Yaskawa INFORM job: SKRZYNIA_4040_180_STOPNI_10B_OLD.JBI

/JOB
//NAME SKRZYNIA_4040_180_STOPNI_10B_OLD
///FOLDERNAME 02-SKRZYNIE_JOBS
//POS
///NPOS 593,593,0,24,0,0
///TOOL 0
///POSTYPE PULSE
///PULSE
C00000=-21231,-51303,42314,2367,6591,-1439
C00001=-12854,-61498,-6635,149088,-29435,16513
C00002=84284,-61498,-6635,149088,14842,16513
C00003=84426,-61498,-62039,149088,14842,16513
C00004=84426,-61498,-83719,149088,14842,16513
C00005=40079,-25830,-61904,72398,37828,17494
C00006=40079,-25830,-61904,72398,37828,17494
C00007=38824,-23395,-60038,72349,38727,17731
C00008=41545,-22667,-59464,70826,37145,18191
C00009=40079,-25830,-61904,72398,37828,17494
C00010=40079,-23879,-31232,97616,36989,2612
C00011=40241,-22903,-30855,97033,36795,2952
C00012=39596,-21803,-29985,96678,37187,3182
C00013=41542,-21522,-29763,96797,35874,3054
C00014=40241,-22903,-30855,97033,36795,2952
C00015=32191,-51498,-15746,88434,42441,22641
C00016=44500,-22967,-34027,49689,40772,15208
C00017=44759,-21950,-33222,49364,40770,15399
C00018=43898,-20603,-32137,49608,41392,15289
C00019=45676,-20288,-31878,48567,40497,15854
C00020=44759,-21950,-33222,49364,40770,15399
C00021=50639,-31838,-53853,40430,42590,20636
C00022=47737,-42531,-47731,84740,46626,-3202
C00023=73324,-51450,-15857,136644,48513,-27329
C00024=28578,-31257,-33285,101874,54895,-3139
C00025=29101,-23166,-41439,93785,52323,3372
C00026=30342,-16402,-40775,90158,51109,6027
C00027=29555,-14242,-38855,90054,51607,6222
C00028=31304,-14182,-38798,89754,50458,6198
C00029=30342,-16402,-40775,90158,51109,6027
C00030=37840,-26567,-47806,97824,39338,5403
C00031=38314,-22656,-45541,96192,38787,6352
C00032=38740,-21749,-44817,95954,38481,6451
C00033=38106,-20505,-43805,95701,38856,6673
C00034=39920,-20274,-43616,95549,37666,6573
C00035=38740,-21749,-44817,95954,38481,6451
C00036=35154,-23288,-28184,89821,43405,2441
C00037=35403,-21021,-26397,89340,43215,2751
C00038=34678,-19569,-25213,89063,43699,2948
C00039=36545,-19419,-25091,89018,42427,2940
C00040=35403,-21021,-26397,89340,43215,2751
C00041=46673,-28267,-59493,36306,49500,22578
C00042=47298,-25083,-54483,36432,48421,22382
C00043=46134,-23276,-53085,36983,49197,22170
C00044=48093,-22778,-52692,35651,48513,22818
C00045=47298,-25083,-54483,36432,48421,22382
C00046=43000,-32780,-49011,53703,41088,15214
C00047=66148,-65994,-55487,105361,28212,-7739
C00048=66148,-65994,-55487,105361,28212,-7739
C00049=59848,-54778,-49507,133915,29212,-10807
C00050=45497,-38347,-41839,114412,32622,-465
C00051=46376,-32635,-46933,102993,29107,5780
C00052=46303,-28031,-46898,97061,28371,8976
C00053=45038,-26161,-45521,96183,29128,9541
C00054=46946,-25787,-45238,96120,27855,9431
C00055=46303,-28031,-46898,97061,28371,8976
C00056=45864,-17128,1685,129467,40696,-9274
C00057=46023,-15894,1830,128891,40053,-8896
C00058=45181,-14790,2774,128176,40341,-8535
C00059=46921,-14545,2986,129317,39465,-9073
C00060=45402,-17127,796,128656,40504,-8810
C00061=42828,-21985,-11573,106778,34538,-1929
C00062=43349,-21404,-11124,106831,34165,-1930
C00063=42250,-19876,-9917,105946,34757,-1485
C00064=44494,-19460,-9583,106781,33302,-1837
C00065=42797,-21858,-11474,106726,34550,-1903
C00066=72417,-67880,-88171,46465,42262,31903
C00067=72417,-67880,-88171,46465,42262,31903
C00068=81480,-74508,-67932,111005,17511,3722
C00069=42492,-36415,-29790,92406,42740,11684
C00070=29699,-14901,-14062,86637,51249,15251
C00071=28921,-12904,-12269,86425,51786,15406
C00072=30978,-12767,-12144,86426,50380,15429
C00073=29506,-17416,-16239,86937,51377,15018
C00074=88410,-69609,-60867,139529,19008,-8209
C00075=62412,-62489,-12046,-12266,17816,34850
C00076=0,-52280,40443,0,6876,0
C00077=-681,-52632,38645,-5695,5489,-631
C00078=-17840,-61498,-6635,-149088,-29435,-16513
C00079=-84284,-61498,-6635,-149088,14842,-16513
C00080=-84426,-61498,-62039,-149088,14842,-16513
C00081=-84426,-61498,-83719,-149088,14842,-16513
C00082=-83351,-27062,-60322,-167360,37385,6517
C00083=-83351,-27062,-60322,-167360,37385,23281
C00084=-45097,-23850,-79932,-76262,26943,-22849
C00085=-48253,-15729,-73342,-71138,25693,-24842
C00086=-50302,-13076,-73239,-65836,25323,-27140
C00087=-49401,-11675,-71961,-66260,25816,-27133
C00088=-50608,-11574,-71867,-65226,25249,-27391
C00089=-49660,-13361,-73494,-66442,25615,-26975
C00090=-48242,-21102,-77802,-73044,25430,-23851
C00091=-42432,-29691,-46140,-101591,34194,-3953
C00092=-40467,-32259,-45349,-89481,35752,-6083
C00093=-35590,-22323,-38089,-87474,43148,-7978
C00094=-34853,-20780,-36847,-87247,43643,-8181
C00095=-37029,-20471,-36594,-86926,42180,-8224
C00096=-35503,-23333,-38886,-87700,43207,-7835
C00097=-41659,-25848,-37197,-61468,39541,-12344
C00098=-42019,-23363,-32043,-63110,38591,-11327
C00099=-41283,-22167,-31102,-63128,39154,-11341
C00100=-43189,-21868,-30866,-62281,38009,-11788
C00101=-40846,-25460,-35158,-62968,39555,-11455
C00102=-39561,-32409,-42051,-71473,38885,-9254
C00103=-88477,-67032,-53890,-125185,13082,17955
C00104=-90715,-66667,-50935,-152816,24533,28486
C00105=-30735,-26920,-32844,-95116,50209,-1071
C00106=-37180,-24683,-31930,-114741,47007,2943
C00107=-36407,-19634,-34656,-109847,45004,-453
C00108=-38352,-16604,-33863,-108521,43129,-1176
C00109=-37479,-14809,-32279,-108169,43576,-1482
C00110=-39395,-14487,-31992,-108361,42368,-1194
C00111=-37253,-18321,-35339,-108644,43916,-1187
C00112=-30948,-19486,-27368,-89515,49970,-2899
C00113=-32453,-17458,-25663,-89179,48933,-3088
C00114=-31896,-16151,-24534,-89028,49305,-3221
C00115=-33527,-16125,-24510,-88960,48196,-3202
C00116=-31291,-18911,-26892,-89421,49733,-2955
C00117=-32789,-14788,-10714,-75998,48642,-1904
C00118=-33953,-13481,-9550,-75758,47902,-2112
C00119=-33380,-12226,-8408,-75670,48319,-2157
C00120=-35020,-12164,-8351,-75529,47228,-2306
C00121=-33300,-14767,-10697,-75957,48300,-1949
C00122=-33300,-14767,-10697,-75957,48300,-1949
C00123=-33901,-13199,-7224,-76945,47663,-1266
C00124=-33178,-11617,-5779,-76815,48184,-1329
C00125=-35129,-11426,-5603,-76688,46886,-1497
C00126=-32900,-14718,-9841,-76444,48459,-1584
C00127=-46324,-38325,-53351,-48650,39022,-16558
C00128=-84678,-53272,-42524,-56273,5220,-14251
C00129=-79949,-57830,-54545,-43165,18800,-25262
C00130=-85199,-63426,-59279,-35356,8253,-25340
C00131=-43240,-40066,-69296,-76804,34492,-13950
C00132=-32352,-24302,-62495,-76398,48702,-17646
C00133=-33867,-19497,-59989,-74208,48202,-18898
C00134=-33043,-17469,-58279,-74274,48770,-19034
C00135=-35172,-17180,-58031,-73305,47532,-19251
C00136=-33150,-20833,-61090,-74721,48572,-18687
C00137=-32525,-19963,-22291,-97454,48417,-2656
C00138=-34479,-17146,-19937,-97221,47013,-2812
C00139=-33716,-15515,-18525,-96928,47480,-3025
C00140=-35357,-15455,-18472,-97073,46375,-2908
C00141=-33341,-18474,-21063,-97306,47817,-2759
C00142=-32838,-10388,7981,-94473,48357,2926
C00143=-33747,-9461,8037,-94117,47673,2571
C00144=-33094,-8062,9377,-93861,48090,2458
C00145=-34952,-7927,9507,-94260,46861,2543
C00146=-33010,-10379,7174,-94037,48174,2591
C00147=-74406,-60637,-53290,-78600,32734,-4861
C00148=-74406,-60637,-53290,-78600,32734,-4861
C00149=-66351,-49775,-22313,-121187,42752,19491
C00150=-38126,-18978,-6321,-103556,42156,4232
C00151=-39485,-17529,-8330,-90200,39091,223
C00152=-38315,-15563,-6658,-89669,39866,-39
C00153=-40130,-15376,-6497,-89855,38637,-21
C00154=-40610,-23081,-12745,-91737,38407,1092
C00155=-82794,-45547,-18103,-153793,26453,27163
///LIMIT ON
C00156=-46099,-67236,-11725,-98004,28606,19827
C00157=275,-40498,62911,330,272,-175
///LIMIT OFF
C00158=-21231,-51303,42314,2367,6591,-1439
C00159=-12854,-61498,-6635,149088,-29435,16513
C00160=84284,-61498,-6635,149088,14842,16513
C00161=84426,-61498,-62039,149088,14842,16513
C00162=84426,-61498,-83719,149088,14842,16513
C00163=40079,-25830,-61904,72398,37828,17494
C00164=43542,-21744,-53414,85694,32141,12908
C00165=43538,-20959,-59091,78847,32551,16732
C00166=40079,-23879,-31232,97616,36989,2612
C00167=41069,-22296,-36683,87871,35939,7163
C00168=41069,-20857,-27994,94343,36275,3375
C00169=40241,-22903,-30855,97033,36795,2952
C00170=44500,-22967,-34027,49689,40772,15208
C00171=37674,-14410,-29425,54908,51799,12689
C00172=37617,-13106,-20810,58248,49229,10178
C00173=44759,-21950,-33222,49364,40770,15399
C00174=50639,-31838,-53853,40430,42590,20636
C00175=47737,-42531,-47731,84740,46626,-3202
C00176=78714,-49092,-28755,133609,38199,-24420
C00177=28578,-31257,-33285,101874,54895,-3139
C00178=29101,-23166,-41439,93785,52323,3372
C00179=31163,-13872,-34138,92103,50752,4440
C00180=31163,-14064,-41434,88282,50498,7326
C00181=30342,-16402,-40775,90158,51109,6027
C00182=37840,-26567,-47806,97824,39338,5403
C00183=38314,-22656,-45541,96192,38787,6352
C00184=39658,-19881,-39017,99036,38353,4498
C00185=39658,-20227,-46296,93241,37598,7980
C00186=38740,-21749,-44817,95954,38481,6451
C00187=35154,-23288,-28184,89821,43405,2441
C00188=36302,-20456,-32356,81251,42995,6506
C00189=36302,-19046,-24537,85721,42698,3608
C00190=35403,-21021,-26397,89340,43215,2751
C00191=46673,-28267,-59493,36306,49500,22578
C00192=35383,-14910,-45807,52457,59655,19882
C00193=35383,-15025,-38926,54776,56903,17744
C00194=47298,-25083,-54483,36432,48421,22382
C00195=43000,-32780,-49011,53703,41088,15214
C00196=90538,-65158,-52413,145953,6697,-22013
C00197=90538,-65158,-52413,145953,6697,-22013
C00198=59848,-54778,-49507,133915,29212,-10807
C00199=45497,-38347,-41839,114412,32622,-465
C00200=46376,-32635,-46933,102993,29107,5780
C00201=38443,-20223,-37840,96971,39567,10287
C00202=38443,-20698,-44956,91660,38993,13539
C00203=46303,-28031,-46898,97061,28371,8976
C00204=45864,-17128,1685,129467,40696,-9274
C00205=38069,-7942,12691,120284,49952,-5070
C00206=38069,-11604,1369,116685,47266,-2469
C00207=45402,-17127,796,128656,40504,-8810
C00208=42828,-21985,-11573,106778,34538,-1929
C00209=33281,-15275,-13406,92642,47209,4970
C00210=33281,-12456,-2996,97026,47894,1870
C00211=42797,-21858,-11474,106726,34550,-1903
C00212=72417,-64226,-72669,53660,37323,27470
C00213=81480,-74508,-67932,111005,17511,3722
C00214=31559,-23192,-27729,97069,50041,14774
C00215=34278,-17590,-29530,108925,47275,14558
C00216=34921,-13948,-26935,108215,46513,15013
C00217=34921,-14719,-34056,104413,45059,17611
C00218=33936,-16225,-25259,110400,48238,13526
C00219=30729,-14807,-22031,91030,50318,16982
C00220=30729,-13019,-13516,94566,50766,14318
C00221=88410,-69609,-60867,139529,19008,-8209
C00222=62412,-62489,-12046,-12266,17816,34850
C00223=0,-52280,40443,0,6876,0
C00224=-681,-52632,38645,-5695,5489,-631
C00225=-17840,-61498,-6635,-149088,-29435,-16513
C00226=-84284,-61498,-6635,-149088,14842,-16513
C00227=-84426,-61498,-62039,-149088,14842,-16513
C00228=-84426,-61498,-83719,-149088,14842,-16513
C00229=-83351,-27062,-60322,-167360,37385,6517
C00230=-83351,-27062,-60322,-167360,37385,23281
C00231=-45097,-23850,-79932,-76262,26943,-22849
C00232=-48253,-15729,-73342,-71138,25693,-24842
C00233=-42869,-6204,-67496,-75794,33821,-25861
C00234=-42869,-3205,-70686,-69723,34977,-29338
C00235=-49660,-13361,-73494,-66442,25615,-26975
C00236=-48242,-21102,-77802,-73044,25430,-23851
C00237=-42432,-29691,-46140,-101591,34194,-3953
C00238=-40467,-32259,-45349,-89481,35752,-6083
C00239=-32032,-15700,-34761,-86363,49905,-9645
C00240=-32032,-14866,-27372,-89947,49973,-6979
C00241=-35503,-23333,-38886,-87700,43207,-7835
C00242=-41659,-25848,-37197,-61468,39541,-12344
C00243=-32550,-13183,-23016,-68651,53358,-8526
C00244=-34023,-12481,-22084,-63241,53452,-9524
C00245=-40846,-25460,-35158,-62968,39555,-11455
C00246=-39561,-32409,-42051,-71473,38885,-9254
C00247=-88477,-67032,-53890,-125185,13082,17955
C00248=-90715,-66667,-50935,-152816,24533,28486
C00249=-30735,-26920,-32844,-95116,50209,-1071
C00250=-37180,-24683,-31930,-114741,47007,2943
C00251=-36407,-19634,-34656,-109847,45004,-453
C00252=-39264,-14095,-28560,-110319,43249,69
C00253=-39254,-14742,-35710,-105973,41627,-2729
C00254=-37253,-18321,-35339,-108644,43916,-1187
C00255=-30948,-19486,-27368,-89515,49970,-2899
C00256=-33188,-17217,-33290,-80523,49125,-7157
C00257=-33231,-16133,-25752,-84153,48705,-4513
C00258=-31291,-18911,-26892,-89421,49733,-2955
C00259=-32789,-14788,-10714,-75998,48642,-1904
C00260=-32456,-10000,-8763,-74569,51725,-2878
C00261=-32456,-7502,814,-78111,50801,-165
C00262=-33300,-14767,-10697,-75957,48300,-1949
C00263=-33300,-14767,-10697,-75957,48300,-1949
C00264=-31039,-7597,-4415,-75714,54029,-1891
C00265=-31745,-5891,1281,-74609,53027,-1007
C00266=-32900,-14718,-9841,-76444,48459,-1584
C00267=-46324,-38325,-53351,-48650,39022,-16558
C00268=-84678,-53272,-42524,-56273,5220,-14251
C00269=-79949,-57830,-54545,-43165,18800,-25262
C00270=-85199,-63426,-59279,-35356,8253,-25340
C00271=-43240,-40066,-69296,-76804,34492,-13950
C00272=-32352,-24302,-62495,-76398,48702,-17646
C00273=-34311,-15084,-43386,-89458,46770,-12174
C00274=-34303,-14562,-49859,-85086,46777,-15220
C00275=-33150,-20833,-61090,-74721,48572,-18687
C00276=-32525,-19963,-22291,-97454,48417,-2656
C00277=-35706,-13608,-12356,-102024,46946,-662
C00278=-35706,-15621,-21438,-97808,45877,-3577
C00279=-33341,-18474,-21063,-97306,47817,-2759
C00280=-32838,-10388,7981,-94473,48357,2926
C00281=-33093,-7396,5806,-90907,49596,566
C00282=-33114,-3922,16616,-94789,50065,3444
C00283=-33010,-10379,7174,-94037,48174,2591
C00284=-73757,-59015,-49060,-81128,30370,-3444
C00285=-66351,-49775,-22313,-115582,40632,19491
C00286=-39230,-13378,9505,-118180,46878,7841
C00287=-45382,-7236,12023,-133378,48537,9962
C00288=-45404,-10871,608,-130166,44845,7725
C00289=-39289,-13633,5656,-114159,44810,6160
C00290=-38323,-13232,3563,-106275,42852,3854
C00291=-39624,-12309,2722,-105485,41613,3229
C00292=-39624,-8328,14658,-110578,43519,6514
C00293=-36264,-16485,7382,-110054,45980,6615
C00294=-44249,-32643,-4456,-118298,43922,12613
C00295=-31781,-48654,10305,-108801,40875,18482
///LIMIT ON
C00296=275,-40498,62911,330,272,-175
///LIMIT OFF
C00297=-21231,-51303,42314,2367,6591,-1439
C00298=-12854,-61498,-6635,149088,-29435,16513
C00299=32880,-72586,-50560,79734,53940,25582
C00300=76664,-93599,-96338,114349,24908,7990
C00301=72545,-76403,-90681,98079,12187,16258
C00302=68435,-42241,-79282,43384,21203,43145
C00303=65057,-16377,-54230,51764,24572,24912
C00304=65057,-16377,-54230,51764,24572,24912
C00305=63338,-14509,-52578,53100,25585,24479
C00306=65493,-13068,-51269,50530,24633,25485
C00307=65057,-16377,-54230,51764,24572,24912
C00308=65057,-15356,-24189,99795,20011,765
C00309=64877,-14372,-23690,98704,20045,1316
C00310=64002,-13489,-22890,98156,20604,1621
C00311=65592,-12702,-22173,98357,19527,1466
C00312=64877,-14372,-23690,98704,20045,1316
C00313=68341,-13254,-25781,29903,31229,25524
C00314=68283,-12212,-24821,29865,31356,25548
C00315=67188,-11145,-23825,30867,31841,25051
C00316=68624,-10377,-23095,29361,31405,25809
C00317=68283,-12212,-24821,29865,31356,25548
C00318=67373,-28813,-51747,26561,36937,27500
C00319=65665,-56911,-59086,75825,31170,1181
C00320=86238,-56758,-47218,93606,16664,-7096
C00321=86238,-56758,-47218,93606,16664,-7096
C00322=58162,-25487,-29222,106212,35121,-6052
C00323=54729,-17550,-36821,90686,35172,3055
C00324=53879,-10723,-35593,84994,35691,6442
C00325=52628,-8898,-33837,85063,36512,6546
C00326=54193,-8333,-33282,84633,35489,6620
C00327=53879,-10723,-35593,84994,35691,6442
C00328=63265,-18185,-41125,95483,22448,4389
C00329=62561,-14368,-38517,92984,22773,5727
C00330=62689,-13396,-37636,92694,22678,5861
C00331=61812,-12400,-36718,92465,23238,6064
C00332=63331,-11679,-36046,92201,22238,6052
C00333=62689,-13396,-37636,92694,22678,5861
C00334=60836,-16142,-22303,87853,25853,3109
C00335=60346,-13901,-20318,87240,26185,3441
C00336=59279,-12702,-19226,86999,26911,3593
C00337=60868,-12050,-18626,86765,25831,3679
C00338=60346,-13901,-20318,87240,26185,3441
C00339=71174,-16943,-50501,16787,44328,31924
C00340=70846,-13961,-45205,17496,43056,31510
C00341=69412,-12602,-43961,18675,43507,30969
C00342=70949,-11616,-43043,17320,43301,31610
C00343=70846,-13961,-45205,17496,43056,31510
C00344=66765,-25643,-43957,33958,30926,25005
C00345=89904,-51519,-74342,14421,36812,44678
C00346=59533,-60921,-66479,83565,41795,11392
C00347=74572,-27669,-34920,136415,14797,-11887
C00348=72479,-21736,-38943,108586,11547,1590
C00349=70901,-17325,-38411,94105,11830,8638
C00350=69318,-15905,-37172,92885,12849,9347
C00351=70820,-15051,-36412,92531,11846,9399
C00352=70901,-17325,-38411,94105,11830,8638
C00353=70927,-7523,10343,151197,29871,-19432
C00354=70517,-6236,10737,150221,29352,-18933
C00355=69462,-5331,11645,148944,29606,-18324
C00356=70849,-4645,12343,150548,29173,-19084
C00357=70402,-7634,9356,150158,29478,-18907
C00358=68660,-13051,-4106,122816,18275,-8999
C00359=68895,-12351,-3471,122899,18094,-9031
C00360=67458,-11121,-2337,120787,18802,-8043
C00361=69212,-10147,-1425,122703,17774,-8922
C00362=68590,-12934,-4000,122687,18305,-8939
C00363=75423,-38775,-29488,68062,11357,11878
C00364=75423,-38775,-29488,68062,11357,11878
C00365=83800,-53438,-37305,103753,25026,-1265
C00366=73693,-43023,-29306,101200,31062,8332
C00367=57182,-8361,13896,122065,42938,1264
C00368=54175,-4244,10116,111777,38351,4895
C00369=53015,-2664,11762,111180,39035,5172
C00370=54334,-2350,12093,111780,38228,4906
C00371=54175,-4244,10116,111777,38351,4895
C00372=89016,-59505,-36896,143842,20811,-11822
C00373=0,-52280,40443,0,6876,0
C00374=-681,-52632,38645,-5695,5489,-631
C00375=-17840,-61498,-6635,-149088,-29435,-16513
C00376=-84284,-61498,-6635,-149088,14842,-16513
C00377=-57949,-92832,-68327,-119114,39180,-13331
C00378=-51160,-78996,-68705,-103851,38676,-21739
C00379=-70129,-12201,-70194,-45988,15849,-32683
C00380=-70861,-4247,-62448,-43170,16032,-33903
C00381=-72229,-1292,-61598,-37253,16795,-36501
C00382=-71164,-286,-60510,-39045,17142,-35862
C00383=-72168,114,-60071,-37345,16819,-36474
C00384=-71747,-1710,-62044,-38091,16943,-36199
C00385=-72086,-8949,-67137,-41785,15362,-34318
C00386=-68226,-19972,-38714,-103620,16923,-1218
C00387=-67549,-22986,-38612,-80975,17520,-9124
C00388=-60286,-14955,-31870,-81576,26630,-9634
C00389=-59206,-13694,-30736,-81541,27366,-9725
C00390=-61026,-12796,-29913,-80837,26167,-9971
C00391=-60502,-15936,-32740,-81790,26471,-9505
C00392=-66711,-16726,-29834,-42060,26790,-21996
C00393=-66477,-14329,-24475,-44917,25565,-20507
C00394=-65503,-13376,-23611,-45716,26132,-20127
C00395=-67048,-12587,-22889,-44009,25442,-20959
C00396=-66009,-16611,-27996,-44380,26285,-20808
C00397=-67084,-23473,-35621,-52822,22843,-18344
C00398=-54372,-63877,-56403,-90862,27079,1323
C00399=-55608,-75012,-34654,-126966,55573,20814
C00400=-55608,-75012,-34654,-126966,55573,20814
C00401=-58069,-20780,-28125,-95622,31565,-134
C00402=-62818,-16895,-25617,-123146,31403,8811
C00403=-60301,-12189,-28106,-114654,29999,4030
C00404=-61167,-8731,-26593,-112607,28768,2985
C00405=-59960,-7252,-25135,-111997,29446,2563
C00406=-61574,-6413,-24296,-112502,28453,2957
C00407=-60636,-10677,-28466,-112685,29164,2987
C00408=-55814,-13636,-22293,-87541,33030,-3263
C00409=-56566,-11270,-20110,-87077,32519,-3496
C00410=-55709,-10167,-19066,-86969,33101,-3589
C00411=-57154,-9687,-18605,-86794,32120,-3632
C00412=-55949,-12989,-21706,-87412,32939,-3330
C00413=-57109,-8613,-4995,-71756,32687,-5152
C00414=-57764,-7017,-3429,-71410,32292,-5358
C00415=-56909,-5946,-2356,-71529,32873,-5273
C00416=-58347,-5433,-1836,-71115,31941,-5534
C00417=-57555,-8453,-4841,-71622,32398,-5235
C00418=-57555,-8453,-4841,-71622,32398,-5235
C00419=-57844,-6749,-1100,-73475,31868,-4209
C00420=-56760,-5394,262,-73573,32605,-4123
C00421=-58439,-4668,1002,-73167,31507,-4396
C00422=-57269,-8513,-4090,-72514,32435,-4729
C00423=-74194,-26905,-45748,-21164,30431,-30370
C00424=-93036,-61583,-83098,-4972,39040,-38907
C00425=-93036,-61583,-83098,-4972,39040,-38907
C00426=-71878,-28414,-61729,-48672,19032,-25171
C00427=-58025,-17185,-56692,-61796,34178,-22014
C00428=-58138,-12270,-53641,-59720,34855,-23185
C00429=-56898,-10637,-52111,-60384,35596,-23031
C00430=-58712,-9745,-51261,-58987,34681,-23500
C00431=-57851,-13714,-54968,-60141,34926,-22995
C00432=-57767,-13689,-16896,-100181,31334,-836
C00433=-58645,-10437,-13885,-99794,30663,-1040
C00434=-57513,-9065,-12573,-99347,31388,-1300
C00435=-58947,-8556,-12078,-99591,30423,-1148
C00436=-58031,-12031,-15383,-99926,31110,-974
C00437=-57646,-4162,14084,-101426,32077,4804
C00438=-58050,-2999,14481,-100683,31666,4357
C00439=-57067,-1784,15765,-100255,32298,4198
C00440=-58672,-1130,16464,-100866,31256,4407
C00441=-57676,-4116,13320,-100600,31921,4338
C00442=-69972,-70945,-58827,-87515,35615,-17
C00443=-69972,-70945,-58827,-87515,35615,-17
C00444=-64053,-11295,342,-114563,25508,8776
C00445=-64305,-9514,-1154,-92513,22236,350
C00446=-62690,-7882,422,-91839,23314,70
C00447=-64201,-7220,1072,-92034,22288,112
C00448=-67149,-14673,-5883,-94845,20391,1413
C00449=-66017,-67071,-29713,-134523,32873,22112
///LIMIT ON
C00450=-46099,-67236,-11725,-98004,28606,19827
C00451=275,-40498,62911,330,272,-175
///LIMIT OFF
C00452=-21231,-51303,42314,2367,6591,-1439
C00453=-12854,-61498,-6635,149088,-29435,16513
C00454=84284,-61498,-6635,149088,14842,16513
C00455=84426,-61498,-62039,149088,14842,16513
C00456=84426,-61498,-83719,149088,14842,16513
C00457=65057,-16377,-54230,51764,24572,24912
C00458=84197,-12836,-45810,-45141,8815,68584
C00459=84197,-12041,-51210,-30828,12194,61758
C00460=65057,-15356,-24189,99795,20011,765
C00461=74080,-15423,-30907,69143,7686,14038
C00462=74080,-14352,-23480,100923,7503,-991
C00463=64877,-14372,-23690,98704,20045,1316
C00464=68341,-13254,-25781,29903,31229,25524
C00465=74439,-11496,-26749,13621,29642,33649
C00466=74439,-10401,-19085,15788,25340,32499
C00467=68283,-12212,-24821,29865,31356,25548
C00468=75452,-19560,-44582,17787,36745,31835
C00469=68183,-44834,-62310,40554,34116,19994
C00470=94103,-63119,-69903,16230,17694,31762
C00471=91219,-55958,-51219,93435,14423,-1742
C00472=58162,-25487,-29222,106212,35121,-6052
C00473=54729,-17550,-36821,90686,35172,3055
C00474=70769,-15160,-35297,83470,11760,4000
C00475=70769,-15377,-40609,67973,12489,11436
C00476=53879,-10723,-35593,84994,35691,6442
C00477=63265,-18185,-41125,95483,22448,4389
C00478=62561,-14368,-38517,92984,22773,5727
C00479=77715,-13962,-33882,144680,4496,-21400
C00480=77806,-14046,-41277,60589,2532,18064
C00481=62689,-13396,-37636,92694,22678,5861
C00482=60836,-16142,-22303,87853,25853,3109
C00483=74678,-16514,-29029,42946,9451,23276
C00484=74678,-15315,-21920,65026,7151,12815
C00485=60346,-13901,-20318,87240,26185,3441
C00486=71174,-16943,-50501,16787,44328,31924
C00487=80494,-13102,-44599,-1731,38384,44653
C00488=80494,-13295,-38861,-1907,34285,44756
C00489=70846,-13961,-45205,17496,43056,31510
C00490=69645,-22678,-41665,30358,30421,26767
C00491=81017,-78801,-66317,80675,7786,2447
C00492=81017,-78801,-66317,80675,7786,2447
C00493=74572,-27669,-34920,136415,14797,-11887
C00494=72479,-21736,-38943,108586,11547,1590
C00495=76162,-15538,-34076,119407,5153,-4143
C00496=76225,-15803,-40874,66675,4586,20654
C00497=70901,-17325,-38411,94105,11830,8638
C00498=70927,-7523,10343,151197,29871,-19432
C00499=75273,-951,23395,164730,33684,-27271
C00500=75257,-4812,11918,163197,28775,-26429
C00501=70402,-7634,9356,150158,29478,-18907
C00502=68660,-13051,-4106,122816,18275,-8999
C00503=75422,-13779,-12311,124767,7049,-10125
C00504=75402,-11409,-3274,143452,10422,-18986
C00505=68590,-12934,-4000,122687,18305,-8939
C00506=83595,-66668,-34414,154325,14846,-28455
C00507=83595,-66668,-34414,154325,14846,-28455
C00508=69137,-30288,-25983,94330,24536,11676
C00509=63448,-5639,10903,136482,36601,-23409
C00510=72869,1541,21011,161481,40400,-32944
C00511=75019,3768,21884,166311,43242,-33805
C00512=75946,3919,31956,167866,49928,-34763
C00513=66712,-14281,-1549,117281,20128,-19574
C00514=72038,-15960,-22039,53337,12147,14456
C00515=72038,-13517,-11162,79650,10019,1887
C00516=70769,-47931,-32777,112213,25945,2479
C00517=17178,-50520,12136,39169,20391,2344
C00518=-681,-52632,38645,-5695,5489,-631
C00519=-17840,-61498,-6635,-149088,-29435,-16513
C00520=-84284,-61498,-6635,-149088,14842,-16513
C00521=-84426,-61498,-62039,-149088,14842,-16513
C00522=-84426,-61498,-83719,-149088,14842,-16513
C00523=-83351,-27062,-60322,-167360,37385,6517
C00524=-83351,-27062,-60322,-167360,37385,23281
C00525=-70129,-12201,-70194,-45988,15849,-32683
C00526=-70861,-4247,-62448,-43170,16032,-33903
C00527=-76882,43,-60950,-14294,14755,-45201
C00528=-76882,3984,-64926,-10429,20329,-47102
C00529=-71747,-1710,-62044,-38091,16943,-36199
C00530=-72086,-8949,-67137,-41785,15362,-34318
C00531=-68226,-19972,-38714,-103620,16923,-1218
C00532=-67549,-22986,-38612,-80975,17520,-9124
C00533=-69143,-15166,-34287,-68804,15212,-14794
C00534=-69143,-14592,-28782,-80821,14459,-8960
C00535=-60502,-15936,-32740,-81790,26471,-9505
C00536=-66711,-16726,-29834,-42060,26790,-21996
C00537=-75652,-13136,-22972,-17539,18443,-33643
C00538=-76393,-11602,-18975,-13556,19574,-34543
C00539=-66009,-16611,-27996,-44380,26285,-20808
C00540=-61601,-28306,-39228,-59626,25389,-15050
C00541=-72315,-63222,-70224,-69600,33305,-10426
C00542=-72315,-63222,-70224,-69600,33305,-10426
C00543=-58069,-20780,-28125,-95622,31565,-134
C00544=-62818,-16895,-25617,-123146,31403,8811
C00545=-60301,-12189,-28106,-114654,29999,4030
C00546=-75089,-9933,-24682,-148597,14783,22922
C00547=-75089,-10642,-34451,-132584,9653,15243
C00548=-60636,-10677,-28466,-112685,29164,2987
C00549=-55814,-13636,-22293,-87541,33030,-3263
C00550=-73301,-16058,-32281,-44459,12702,-22095
C00551=-73339,-15052,-25249,-60236,10249,-14543
C00552=-55949,-12989,-21706,-87412,32939,-3330
C00553=-57109,-8613,-4995,-71756,32687,-5152
C00554=-71674,-10355,-9102,-48278,15013,-17468
C00555=-71670,-8088,-356,-62615,12652,-10541
C00556=-57555,-8453,-4841,-71622,32398,-5235
C00557=-57555,-8453,-4841,-71622,32398,-5235
C00558=-73349,-10209,-7254,-46090,12597,-18565
C00559=-73349,-7867,1452,-63091,10217,-10432
C00560=-57269,-8513,-4090,-72514,32435,-4729
C00561=-74194,-26905,-45748,-21164,30431,-30370
C00562=-76007,-77202,-67157,-59280,11041,-11579
C00563=-76006,-77203,-67157,-59281,11043,-11581
C00564=-53398,-42726,-55849,-45492,34374,-18069
C00565=-71878,-28414,-61729,-48672,19032,-25171
C00566=-58025,-17185,-56692,-61796,34178,-22014
C00567=-77553,-14661,-43008,-35465,5780,-31120
C00568=-77553,-14004,-50514,-17997,10868,-39389
C00569=-57851,-13714,-54968,-60141,34926,-22995
C00570=-57767,-13689,-16896,-100181,31334,-836
C00571=-74769,-11126,-10073,-142523,13426,19686
C00572=-74753,-12848,-17783,-130765,10301,14051
C00573=-58031,-12031,-15383,-99926,31110,-974
C00574=-57646,-4162,14084,-101426,32077,4804
C00575=-72179,-7124,6017,-115427,12582,9833
C00576=-72179,-4103,15503,-129018,15105,16401
C00577=-57676,-4116,13320,-100600,31921,4338
C00578=-68334,-63389,-52515,-83837,33201,-1739
C00579=-68334,-63389,-52515,-83837,33201,-1739
C00580=-64053,-11295,342,-114563,25508,8776
C00581=-76017,6008,33610,-165984,45639,36413
C00582=-74239,7065,32887,-163372,44700,35065
C00583=-74142,3045,20239,-161993,39159,34198
C00584=-75119,4045,29308,-164063,44402,35406
C00585=-79833,-9558,5437,-165750,9898,43323
C00586=-75231,-7555,5870,-137998,10766,30530
C00587=-75231,-3987,16941,-149127,14978,35883
C00588=-77761,-13214,8113,-156332,15145,39163
C00589=-65551,-48104,-28924,-114827,24376,11665
C00590=-51220,-46814,3045,-130057,64886,23876
///LIMIT ON
C00591=-46099,-67236,-11725,-98004,28606,19827
C00592=275,-40498,62911,330,272,-175
///LIMIT OFF
BC00000=375059
BC00001=421503
BC00002=401943
BC00003=375374
BC00004=375374
BC00005=386710
BC00006=386710
BC00007=386710
BC00008=386710
BC00009=386710
BC00010=386710
BC00011=386710
BC00012=386710
BC00013=386710
BC00014=386710
BC00015=396872
BC00016=386710
BC00017=386710
BC00018=386710
BC00019=386710
BC00020=386710
BC00021=386710
BC00022=389814
BC00023=471786
BC00024=514090
BC00025=514090
BC00026=514086
BC00027=514086
BC00028=514086
BC00029=514086
BC00030=562496
BC00031=562452
BC00032=562452
BC00033=562452
BC00034=562452
BC00035=562452
BC00036=562452
BC00037=562452
BC00038=562452
BC00039=562452
BC00040=562452
BC00041=594236
BC00042=594236
BC00043=594184
BC00044=594184
BC00045=594236
BC00046=560408
BC00047=555998
BC00048=669671
BC00049=691880
BC00050=691880
BC00051=691880
BC00052=691880
BC00053=691880
BC00054=691880
BC00055=691880
BC00056=784046
BC00057=784046
BC00058=784046
BC00059=784046
BC00060=784046
BC00061=821134
BC00062=821134
BC00063=821134
BC00064=821134
BC00065=821134
BC00066=665295
BC00067=757461
BC00068=745890
BC00069=709907
BC00070=709907
BC00071=709907
BC00072=709907
BC00073=709907
BC00074=745890
BC00075=625968
BC00076=597988
BC00077=426820
BC00078=417754
BC00079=375374
BC00080=375374
BC00081=375374
BC00082=429001
BC00083=428186
BC00084=443593
BC00085=443593
BC00086=443591
BC00087=443591
BC00088=443591
BC00089=443591
BC00090=443591
BC00091=393487
BC00092=393487
BC00093=393487
BC00094=393487
BC00095=393487
BC00096=393487
BC00097=393487
BC00098=393487
BC00099=393487
BC00100=393487
BC00101=393487
BC00102=393487
BC00103=393487
BC00104=522946
BC00105=522946
BC00106=522946
BC00107=522946
BC00108=522946
BC00109=522946
BC00110=522946
BC00111=522946
BC00112=522946
BC00113=522946
BC00114=522946
BC00115=522946
BC00116=522946
BC00117=522946
BC00118=522946
BC00119=522946
BC00120=522946
BC00121=522946
BC00122=565910
BC00123=565910
BC00124=565910
BC00125=565910
BC00126=565910
BC00127=563514
BC00128=551555
BC00129=551555
BC00130=701230
BC00131=706904
BC00132=706904
BC00133=706904
BC00134=706904
BC00135=706904
BC00136=706904
BC00137=799070
BC00138=799070
BC00139=799070
BC00140=799070
BC00141=799070
BC00142=799070
BC00143=799070
BC00144=799070
BC00145=799070
BC00146=799070
BC00147=635036
BC00148=727202
BC00149=699743
BC00150=699743
BC00151=699743
BC00152=699743
BC00153=699743
BC00154=699743
BC00155=699743
BC00156=665064
BC00157=408992
BC00158=375059
BC00159=421503
BC00160=401943
BC00161=375374
BC00162=375374
BC00163=386710
BC00164=386710
BC00165=386710
BC00166=386710
BC00167=386710
BC00168=386710
BC00169=386710
BC00170=386710
BC00171=386710
BC00172=386710
BC00173=386710
BC00174=386710
BC00175=389814
BC00176=492157
BC00177=514090
BC00178=514090
BC00179=514086
BC00180=514086
BC00181=514086
BC00182=562496
BC00183=562452
BC00184=562452
BC00185=562452
BC00186=562452
BC00187=562452
BC00188=562452
BC00189=562452
BC00190=562452
BC00191=594236
BC00192=594236
BC00193=594236
BC00194=594236
BC00195=560408
BC00196=549248
BC00197=623644
BC00198=691880
BC00199=691880
BC00200=691880
BC00201=691880
BC00202=691880
BC00203=691880
BC00204=784046
BC00205=784043
BC00206=784043
BC00207=784046
BC00208=821134
BC00209=821134
BC00210=821134
BC00211=821134
BC00212=665295
BC00213=744345
BC00214=744345
BC00215=744345
BC00216=744345
BC00217=744345
BC00218=744345
BC00219=744345
BC00220=744345
BC00221=749235
BC00222=625363
BC00223=556260
BC00224=380737
BC00225=417754
BC00226=375374
BC00227=375374
BC00228=375374
BC00229=429001
BC00230=428186
BC00231=443593
BC00232=443593
BC00233=443591
BC00234=443591
BC00235=443591
BC00236=443591
BC00237=393487
BC00238=393487
BC00239=393487
BC00240=393487
BC00241=393487
BC00242=393487
BC00243=393487
BC00244=393487
BC00245=393487
BC00246=393487
BC00247=393487
BC00248=522946
BC00249=522946
BC00250=522946
BC00251=522946
BC00252=522946
BC00253=522946
BC00254=522946
BC00255=522946
BC00256=522946
BC00257=522946
BC00258=522946
BC00259=522946
BC00260=522946
BC00261=522946
BC00262=522946
BC00263=565910
BC00264=565910
BC00265=565910
BC00266=565910
BC00267=563514
BC00268=551555
BC00269=551555
BC00270=701230
BC00271=706904
BC00272=706904
BC00273=706904
BC00274=706904
BC00275=706904
BC00276=799070
BC00277=799070
BC00278=799070
BC00279=799070
BC00280=799070
BC00281=799070
BC00282=799070
BC00283=799070
BC00284=626135
BC00285=699743
BC00286=710175
BC00287=710175
BC00288=710175
BC00289=710175
BC00290=719551
BC00291=719551
BC00292=719551
BC00293=719551
BC00294=708451
BC00295=648955
BC00296=455075
BC00297=375059
BC00298=421503
BC00299=450455
BC00300=443143
BC00301=386198
BC00302=386198
BC00303=386710
BC00304=386710
BC00305=386710
BC00306=386710
BC00307=386710
BC00308=386710
BC00309=386710
BC00310=386710
BC00311=386710
BC00312=386710
BC00313=386710
BC00314=386710
BC00315=386710
BC00316=386710
BC00317=386710
BC00318=386710
BC00319=388593
BC00320=388593
BC00321=468229
BC00322=514090
BC00323=514090
BC00324=514086
BC00325=514086
BC00326=514086
BC00327=514086
BC00328=562496
BC00329=562452
BC00330=562452
BC00331=562452
BC00332=562452
BC00333=562452
BC00334=562452
BC00335=562452
BC00336=562452
BC00337=562452
BC00338=562452
BC00339=594236
BC00340=594236
BC00341=594184
BC00342=594184
BC00343=594236
BC00344=560408
BC00345=560408
BC00346=682684
BC00347=691880
BC00348=691880
BC00349=691880
BC00350=691880
BC00351=691880
BC00352=691880
BC00353=784046
BC00354=784046
BC00355=784046
BC00356=784046
BC00357=784046
BC00358=821134
BC00359=821134
BC00360=821134
BC00361=821134
BC00362=821134
BC00363=636802
BC00364=728968
BC00365=735310
BC00366=802073
BC00367=802073
BC00368=802073
BC00369=802073
BC00370=802073
BC00371=802073
BC00372=817725
BC00373=657110
BC00374=472903
BC00375=509920
BC00376=467540
BC00377=497868
BC00378=497868
BC00379=535759
BC00380=535759
BC00381=535757
BC00382=535757
BC00383=535757
BC00384=535757
BC00385=535757
BC00386=485653
BC00387=485653
BC00388=485653
BC00389=485653
BC00390=485653
BC00391=485653
BC00392=485653
BC00393=485653
BC00394=485653
BC00395=485653
BC00396=485653
BC00397=485653
BC00398=485653
BC00399=485653
BC00400=601945
BC00401=615112
BC00402=615112
BC00403=615112
BC00404=615112
BC00405=615112
BC00406=615112
BC00407=615112
BC00408=615112
BC00409=615112
BC00410=615112
BC00411=615112
BC00412=615112
BC00413=615112
BC00414=615112
BC00415=615112
BC00416=615112
BC00417=615112
BC00418=658076
BC00419=658076
BC00420=658076
BC00421=658076
BC00422=658076
BC00423=655680
BC00424=655680
BC00425=765678
BC00426=799070
BC00427=799070
BC00428=799070
BC00429=799070
BC00430=799070
BC00431=799070
BC00432=799070
BC00433=799070
BC00434=799070
BC00435=799070
BC00436=799070
BC00437=799070
BC00438=799070
BC00439=799070
BC00440=799070
BC00441=799070
BC00442=736060
BC00443=824347
BC00444=791909
BC00445=791909
BC00446=791909
BC00447=791909
BC00448=791909
BC00449=791909
BC00450=757230
BC00451=501158
BC00452=467225
BC00453=513669
BC00454=494109
BC00455=467540
BC00456=467540
BC00457=478876
BC00458=478876
BC00459=478876
BC00460=478876
BC00461=478876
BC00462=478876
BC00463=478876
BC00464=478876
BC00465=478876
BC00466=478876
BC00467=478876
BC00468=478876
BC00469=479530
BC00470=502776
BC00471=571156
BC00472=606256
BC00473=606256
BC00474=606252
BC00475=606252
BC00476=606252
BC00477=654662
BC00478=654618
BC00479=654618
BC00480=654618
BC00481=654618
BC00482=654618
BC00483=654618
BC00484=654618
BC00485=654618
BC00486=686402
BC00487=686402
BC00488=686402
BC00489=686402
BC00490=652574
BC00491=654591
BC00492=763025
BC00493=784046
BC00494=784046
BC00495=784046
BC00496=784046
BC00497=784046
BC00498=784046
BC00499=784043
BC00500=784043
BC00501=784046
BC00502=821134
BC00503=821134
BC00504=821134
BC00505=821134
BC00506=720655
BC00507=777239
BC00508=814624
BC00509=805198
BC00510=810577
BC00511=810577
BC00512=810577
BC00513=810577
BC00514=823729
BC00515=823729
BC00516=813320
BC00517=702447
BC00518=518986
BC00519=509920
BC00520=467540
BC00521=467540
BC00522=467540
BC00523=521167
BC00524=520352
BC00525=535759
BC00526=535759
BC00527=535757
BC00528=535757
BC00529=535757
BC00530=535757
BC00531=485653
BC00532=485653
BC00533=485653
BC00534=485653
BC00535=485653
BC00536=485653
BC00537=485653
BC00538=485653
BC00539=485653
BC00540=485653
BC00541=485653
BC00542=600333
BC00543=615112
BC00544=615112
BC00545=615112
BC00546=615112
BC00547=615112
BC00548=615112
BC00549=615112
BC00550=615112
BC00551=615112
BC00552=615112
BC00553=615112
BC00554=615112
BC00555=615112
BC00556=615112
BC00557=658076
BC00558=658076
BC00559=658076
BC00560=658076
BC00561=655680
BC00562=656245
BC00563=762546
BC00564=762546
BC00565=799070
BC00566=799070
BC00567=799070
BC00568=799070
BC00569=799070
BC00570=799070
BC00571=799070
BC00572=799070
BC00573=799070
BC00574=799070
BC00575=799070
BC00576=799070
BC00577=799070
BC00578=722449
BC00579=802864
BC00580=791909
BC00581=807068
BC00582=807068
BC00583=807068
BC00584=807068
BC00585=807068
BC00586=807068
BC00587=807068
BC00588=807068
BC00589=799597
BC00590=784137
BC00591=739235
BC00592=547241
///POSTYPE BASE
///RECTAN
///RCONF 1,0,0,0,0,0,0,0,0,0,0,0,0,0,0,0,0,0,0,0,0,0,0,0
P00006=0.000,0.000,0.000,0.0000,0.0000,0.0000
///RCONF 0,0,0,0,0,0,0,0,0,0,0,0,0,0,0,0,0,0,0,0,0,0,0,0
P00056=0.000,0.000,5.000,0.0000,0.0000,0.0000
///RCONF 1,0,0,0,0,0,0,0,0,0,0,0,0,0,0,0,0,0,0,0,0,0,0,0
P00301=0.046,-2.112,7.779,0.0000,0.0000,0.0000
P00302=-0.180,-2.409,6.326,0.0000,0.0000,0.0000
///RCONF 0,0,0,0,0,0,0,0,0,0,0,0,0,0,0,0,0,0,0,0,0,0,0,0
P00303=-0.004,-1.437,-4.584,0.0000,0.0000,0.0000
P00304=0.028,-1.666,-4.234,0.0000,0.0000,0.0000
P00305=-0.003,-1.920,-3.501,0.0000,0.0000,0.0000
P00306=0.015,-2.252,-3.054,0.0000,0.0000,0.0000
P00307=0.019,-2.151,-5.077,0.0000,0.0000,0.0000
P00308=-0.003,-2.092,-4.888,0.0000,0.0000,0.0000
P00309=-0.040,-2.205,-4.992,0.0000,0.0000,0.0000
P00310=-0.006,-2.490,-5.925,0.0000,0.0000,0.0000
P00312=-0.032,2.202,-7.632,0.0000,0.0000,0.0000
P00351=13.563,-0.027,-0.653,0.0000,0.0000,0.0000
P00352=13.252,-0.027,-0.827,0.0000,0.0000,0.0000
P00353=10.971,-0.082,0.776,0.0000,0.0000,0.0000
P00354=-0.024,2.508,-1.824,0.0000,0.0000,0.0000
P00355=-0.001,2.528,-1.131,0.0000,0.0000,0.0000
P00356=-0.034,2.921,-0.262,0.0000,0.0000,0.0000
P00357=0.003,3.386,-0.091,0.0000,0.0000,0.0000
P00358=0.014,3.037,-0.020,0.0000,0.0000,0.0000
P00359=-0.005,2.731,0.912,0.0000,0.0000,0.0000
P00360=-0.011,3.412,0.438,0.0000,0.0000,0.0000
P00362=0.014,2.784,0.148,0.0000,0.0000,0.0000
//INST
///DATE 2025/03/26 10:36
///ATTR SC,RW
///GROUP1 RB1,BS1
NOP
CALL JOB:MOVE_INTO_TUNNEL
MOVJ C00000 BC00000 VJ=10.00
MOVJ C00001 BC00001 VJ=10.00
MOVJ C00002 BC00002 VJ=10.00
COMM MOVJ C00003 BC00003 VJ=10.00
COMM MOVJ C00004 BC00004 VJ=10.00
COMM '------------------------
COMM 'W29.2
COMM '------------------------
COMM MOVL C00005 BC00005 V=500.0
COMM '------------------------
COMM 'W63.5
COMM '------------------------
COMM SFTOF
COMM MOVL C00006 BC00006 V=166.7 PL=0
COMM REFP 3 C00007 BC00007
COMM CALL JOB:SEARCH-R1
COMM IMOV P0056 V=50.0 PL=0
COMM SET P0301 P0006
COMM SFTON P0301
COMM REFP 3 C00008 BC00008
COMM CALL JOB:SEARCH-R1
COMM SET P0301 P0006
COMM SFTON P0301
COMM MOVL C00009 BC00009 V=166.7 PL=0
COMM SFTOF
COMM MOVL C00010 BC00010 V=500.0
COMM MOVL C00011 BC00011 V=166.7 PL=0
COMM REFP 3 C00012 BC00012
COMM CALL JOB:SEARCH-R1
COMM IMOV P0056 V=50.0 PL=0
COMM SET P0302 P0006
COMM SFTON P0302
COMM REFP 3 C00013 BC00013
COMM CALL JOB:SEARCH-R1
COMM SET P0302 P0006
COMM SFTON P0302
COMM MOVL C00014 BC00014 V=166.7 PL=0
SFTOF
MOVJ C00015 BC00015 VJ=10.00
MOVL C00016 BC00016 V=500.0
MOVL C00017 BC00017 V=166.7 PL=0
REFP 3 C00018 BC00018
CALL JOB:SEARCH-R1
IMOV P0056 V=50.0 PL=0
SET P0303 P0006
SFTON P0303
REFP 3 C00019 BC00019
CALL JOB:SEARCH-R1
SET P0303 P0006
SFTON P0303
SFTOF
MOVL C00020 BC00020 V=166.7 PL=0
MOVL C00021 BC00021 V=500.0
MOVJ C00022 BC00022 VJ=30.00
MOVJ C00023 BC00023 VJ=30.00
MOVJ C00024 BC00024 VJ=30.00
MOVL C00025 BC00025 V=500.0
'------------------------
'W29.14
'------------------------
MOVL C00026 BC00026 V=166.7 PL=0
REFP 3 C00027 BC00027
CALL JOB:SEARCH-R1
IMOV P0056 V=23.0 PL=0
SET P0304 P0006
SFTON P0304
REFP 3 C00028 BC00028
CALL JOB:SEARCH-R1
SET P0304 P0006
SFTON P0304
MOVL C00029 BC00029 V=66.7 PL=0
SFTOF
'PRZEJAZD
MOVL C00030 BC00030 V=500.0
MOVL C00031 BC00031 V=500.0
'------------------------
'W63.17
'------------------------
MOVL C00032 BC00032 V=166.7 PL=0
REFP 3 C00033 BC00033
CALL JOB:SEARCH-R1
IMOV P0056 V=23.0 PL=0
SET P0305 P0006
SFTON P0305
REFP 3 C00034 BC00034
CALL JOB:SEARCH-R1
SET P0305 P0006
SFTON P0305
MOVL C00035 BC00035 V=166.7 PL=0
SFTOF
MOVL C00036 BC00036 V=500.0
MOVL C00037 BC00037 V=166.7
REFP 3 C00038 BC00038
CALL JOB:SEARCH-R1
IMOV P0056 V=23.0 PL=0
SET P0306 P0006
SFTON P0306
REFP 3 C00039 BC00039
CALL JOB:SEARCH-R1
SET P0306 P0006
SFTON P0306
MOVL C00040 BC00040 V=166.7 PL=0
'PRZEJAZD
MOVL C00041 BC00041 V=500.0
MOVL C00042 BC00042 V=166.7
REFP 3 C00043 BC00043
CALL JOB:SEARCH-R1
IMOV P0056 V=23.0 PL=0
SET P0307 P0006
SFTON P0307
REFP 3 C00044 BC00044
CALL JOB:SEARCH-R1
SET P0307 P0006
SFTON P0307
MOVL C00045 BC00045 V=166.7 PL=0
SFTOF
MOVJ C00046 BC00046 VJ=20.00
MOVJ C00047 BC00047 VJ=20.00
MOVJ C00048 BC00048 VJ=30.00
MOVJ C00049 BC00049 VJ=30.00
MOVJ C00050 BC00050 VJ=30.00
MOVL C00051 BC00051 V=500.0
'------------------------
'W63.20
'------------------------
MOVL C00052 BC00052 V=166.7 PL=0
REFP 3 C00053 BC00053
CALL JOB:SEARCH-R1
IMOV P0056 V=23.0 PL=0
SET P0308 P0006
SFTON P0308
REFP 3 C00054 BC00054
CALL JOB:SEARCH-R1
SET P0308 P0006
SFTON P0308
MOVL C00055 BC00055 V=166.7 PL=0
SFTOF
COMM 'PRZEJAZD
COMM MOVL C00056 BC00056 V=500.0
COMM '------------------------
COMM 'W63.23
COMM '------------------------
COMM MOVL C00057 BC00057 V=166.7 PL=0
COMM REFP 3 C00058 BC00058
COMM CALL JOB:SEARCH-R1
COMM IMOV P0056 V=23.0 PL=0
COMM SET P0309 P0006
COMM SFTON P0309
COMM REFP 3 C00059 BC00059
COMM CALL JOB:SEARCH-R1
COMM SET P0309 P0006
COMM SFTON P0309
COMM MOVL C00060 BC00060 V=250.0 PL=0
COMM SFTOF
COMM MOVL C00061 BC00061 V=500.0
COMM MOVL C00062 BC00062 V=166.7 PL=0
COMM REFP 3 C00063 BC00063
COMM CALL JOB:SEARCH-R1
COMM IMOV P0056 V=23.0 PL=0
COMM SET P0310 P0006
COMM SFTON P0310
COMM REFP 3 C00064 BC00064
COMM CALL JOB:SEARCH-R1
COMM SET P0310 P0006
COMM SFTON P0310
COMM MOVL C00065 BC00065 V=250.0 PL=0
COMM SFTOF
MOVL C00066 BC00066 V=500.0
MOVL C00067 BC00067 V=500.0
MOVL C00068 BC00068 V=500.0
MOVL C00069 BC00069 V=333.3
'------------------------
'W29.29
'------------------------
MOVL C00070 BC00070 V=166.7 PL=0
REFP 3 C00071 BC00071
CALL JOB:SEARCH-R1
IMOV P0056 V=23.0 PL=0
SET P0312 P0006
SFTON P0312
REFP 3 C00072 BC00072
CALL JOB:SEARCH-R1
SET P0312 P0006
SFTON P0312
MOVL C00073 BC00073 V=250.0 PL=0
SFTOF
'PRZEJAZD
MOVL C00074 BC00074 V=333.3
'PRZEJAZD
MOVJ C00075 BC00075 VJ=30.00
MOVJ C00076 BC00076 VJ=20.00
MOVJ C00077 BC00077 VJ=50.00
MOVJ C00078 BC00078 VJ=20.00
MOVJ C00079 BC00079 VJ=10.00
MOVJ C00080 BC00080 VJ=20.00
MOVJ C00081 BC00081 VJ=20.00
'------------------------
'W28.2
'------------------------
MOVJ C00082 BC00082 VJ=10.00
MOVJ C00083 BC00083 VJ=10.00
MOVL C00084 BC00084 V=500.0
MOVL C00085 BC00085 V=500.0
'------------------------
'W62.5
'------------------------
MOVL C00086 BC00086 V=166.7 PL=0
REFP 3 C00087 BC00087
CALL JOB:SEARCH-R1
IMOV P0056 V=23.0 PL=0
SET P0351 P0006
SFTON P0351
REFP 3 C00088 BC00088
CALL JOB:SEARCH-R1
SET P0351 P0006
SFTON P0351
MOVL C00089 BC00089 V=250.0 PL=0
SFTOF
'PRZEJAZD
MOVL C00090 BC00090 V=500.0
MOVL C00091 BC00091 V=500.0
MOVL C00092 BC00092 V=500.0
MOVL C00093 BC00093 V=166.7 PL=0
REFP 3 C00094 BC00094
CALL JOB:SEARCH-R1
IMOV P0056 V=23.0 PL=0
SET P0352 P0006
SFTON P0352
REFP 3 C00095 BC00095
CALL JOB:SEARCH-R1
SET P0352 P0006
SFTON P0352
MOVL C00096 BC00096 V=250.0 PL=0
SFTOF
MOVL C00097 BC00097 V=500.0
'------------------------
'W29.8
'------------------------
MOVL C00098 BC00098 V=166.7 PL=0
REFP 3 C00099 BC00099
CALL JOB:SEARCH-R1
IMOV P0056 V=23.0 PL=0
SET P0353 P0006
SFTON P0353
REFP 3 C00100 BC00100
CALL JOB:SEARCH-R1
SET P0353 P0006
SFTON P0353
MOVL C00101 BC00101 V=250.0 PL=0
SFTOF
MOVL C00102 BC00102 V=500.0
'PRZEJAZD
MOVL C00103 BC00103 V=500.0
MOVJ C00104 BC00104 VJ=20.00
MOVL C00105 BC00105 V=500.0
MOVL C00106 BC00106 V=500.0
MOVL C00107 BC00107 V=500.0
'------------------------
'W29.11
'------------------------
MOVL C00108 BC00108 V=166.7 PL=0
REFP 3 C00109 BC00109
CALL JOB:SEARCH-R1
IMOV P0056 V=23.0 PL=0
SET P0354 P0006
SFTON P0354
REFP 3 C00110 BC00110
CALL JOB:SEARCH-R1
SET P0354 P0006
SFTON P0354
MOVL C00111 BC00111 V=250.0 PL=0
SFTOF
'PRZEJAZD
MOVL C00112 BC00112 V=500.0
'------------------------
'W29.14
'------------------------
MOVL C00113 BC00113 V=166.7 PL=0
REFP 3 C00114 BC00114
CALL JOB:SEARCH-R1
IMOV P0056 V=23.0 PL=0
SET P0355 P0006
SFTON P0355
REFP 3 C00115 BC00115
CALL JOB:SEARCH-R1
SET P0355 P0006
SFTON P0355
MOVL C00116 BC00116 V=250.0 PL=0
SFTOF
'PRZEJAZD
MOVL C00117 BC00117 V=500.0
'------------------------
'W63.17
'------------------------
MOVL C00118 BC00118 V=166.7 PL=0
REFP 3 C00119 BC00119
CALL JOB:SEARCH-R1
IMOV P0056 V=23.0 PL=0
SET P0356 P0006
SFTON P0356
REFP 3 C00120 BC00120
CALL JOB:SEARCH-R1
SET P0356 P0006
SFTON P0356
MOVL C00121 BC00121 V=250.0 PL=0
SFTOF
MOVL C00122 BC00122 V=500.0
MOVL C00123 BC00123 V=166.7 PL=0
REFP 3 C00124 BC00124
CALL JOB:SEARCH-R1
IMOV P0056 V=23.0 PL=0
SET P0357 P0006
SFTON P0357
REFP 3 C00125 BC00125
CALL JOB:SEARCH-R1
SET P0357 P0006
SFTON P0357
MOVL C00126 BC00126 V=250.0 PL=0
SFTOF
'PRZEJAZD
MOVL C00127 BC00127 V=500.0
MOVJ C00128 BC00128 VJ=30.00
MOVJ C00129 BC00129 VJ=30.00
MOVJ C00130 BC00130 VJ=30.00
MOVL C00131 BC00131 V=500.0
MOVL C00132 BC00132 V=500.0
'------------------------
'W62.20
'------------------------
MOVL C00133 BC00133 V=166.7 PL=0
REFP 3 C00134 BC00134
CALL JOB:SEARCH-R1
IMOV P0056 V=23.0 PL=0
SET P0358 P0006
SFTON P0358
REFP 3 C00135 BC00135
CALL JOB:SEARCH-R1
SET P0358 P0006
SFTON P0358
MOVL C00136 BC00136 V=250.0 PL=0
SFTOF
COMM 'PRZEJAZD
COMM MOVL C00137 BC00137 V=500.0
COMM '------------------------
COMM 'W63.23
COMM '------------------------
COMM MOVL C00138 BC00138 V=166.7 PL=0
COMM REFP 3 C00139 BC00139
COMM CALL JOB:SEARCH-R1
COMM IMOV P0056 V=23.0 PL=0
COMM SET P0359 P0006
COMM SFTON P0359
COMM REFP 3 C00140 BC00140
COMM CALL JOB:SEARCH-R1
COMM SET P0359 P0006
COMM SFTON P0359
COMM MOVL C00141 BC00141 V=250.0 PL=0
COMM MOVL C00142 BC00142 V=500.0
COMM '------------------------
COMM 'W29.29
COMM '------------------------
COMM MOVL C00143 BC00143 V=166.7 PL=0
COMM REFP 3 C00144 BC00144
COMM CALL JOB:SEARCH-R1
COMM IMOV P0056 V=23.0 PL=0
COMM SET P0360 P0006
COMM SFTON P0360
COMM REFP 3 C00145 BC00145
COMM CALL JOB:SEARCH-R1
COMM SET P0360 P0006
COMM SFTON P0360
COMM MOVL C00146 BC00146 V=250.0 PL=0
COMM SFTOF
COMM 'PRZEJAZD
COMM SFTOF
COMM '------------------------
COMM 'W29.32
COMM '------------------------
COMM 'PRZEJAZD
MOVL C00147 BC00147 V=500.0
MOVL C00148 BC00148 V=500.0
MOVJ C00149 BC00149 VJ=10.00
MOVL C00150 BC00150 V=416.7
MOVL C00151 BC00151 V=166.7 PL=0
REFP 3 C00152 BC00152
CALL JOB:SEARCH-R1
IMOV P0056 V=23.0 PL=0
SET P0362 P0006
SFTON P0362
REFP 3 C00153 BC00153
CALL JOB:SEARCH-R1
SET P0362 P0006
SFTON P0362
MOVL C00154 BC00154 V=250.0 PL=0
SFTOF
MOVJ C00155 BC00155 VJ=20.00
MOVJ C00156 BC00156 VJ=30.00
MOVJ C00157 BC00157 VJ=30.00
'KONIEC SEARCH WEW STRONA
MOVJ C00158 BC00158 VJ=30.00
MOVJ C00159 BC00159 VJ=20.00
MOVJ C00160 BC00160 VJ=10.00
MOVJ C00161 BC00161 VJ=20.00
MOVJ C00162 BC00162 VJ=20.00
'------------------------
'W29.2
'------------------------
MOVL C00163 BC00163 V=500.0
'------------------------
'W63.5
MACRO1 MJ#(0) ARGF9
'------------------------
SFTOF
SFTON P0301
MOVL C00164 BC00164 V=166.7 PL=0
ARCON
MOVL C00165 BC00165 V=10.0
ARCOF
SFTOF
MOVL C00166 BC00166 V=500.0
SFTON P0302
MOVL C00167 BC00167 V=166.7 PL=0
ARCON
MOVL C00168 BC00168 V=10.0
ARCOF
MOVL C00169 BC00169 V=166.7 PL=0
SFTOF
MOVL C00170 BC00170 V=500.0
SFTON P0303
MOVL C00171 BC00171 V=166.7 PL=0
ARCON
MOVL C00172 BC00172 V=10.0
ARCOF
SFTOF
MOVL C00173 BC00173 V=166.7 PL=0
MOVL C00174 BC00174 V=500.0
MOVJ C00175 BC00175 VJ=30.00
MOVJ C00176 BC00176 VJ=30.00
MOVJ C00177 BC00177 VJ=30.00
MOVL C00178 BC00178 V=500.0
'------------------------
'W29.14
'------------------------
SFTON P0304
MOVL C00179 BC00179 V=166.7 PL=0
ARCON
MOVL C00180 BC00180 V=10.0
ARCOF
MOVL C00181 BC00181 V=166.7 PL=0
SFTOF
'PRZEJAZD
MOVL C00182 BC00182 V=500.0
MOVL C00183 BC00183 V=500.0
'------------------------
'W63.17
'------------------------
SFTON P0305
MOVL C00184 BC00184 V=166.7 PL=0
ARCON
MOVL C00185 BC00185 V=10.0
ARCOF
MOVL C00186 BC00186 V=166.7 PL=0
SFTOF
MOVL C00187 BC00187 V=500.0
SFTON P0306
MOVL C00188 BC00188 V=166.7
ARCON
MOVL C00189 BC00189 V=10.0
ARCOF
MOVL C00190 BC00190 V=166.7 PL=0
SFTOF
'PRZEJAZD
MOVL C00191 BC00191 V=500.0
SFTON P0307
MOVL C00192 BC00192 V=166.7
ARCON
MOVL C00193 BC00193 V=10.0
ARCOF
MOVL C00194 BC00194 V=166.7 PL=0
SFTOF
MOVJ C00195 BC00195 VJ=20.00
MOVJ C00196 BC00196 VJ=20.00
MOVJ C00197 BC00197 VJ=30.00
MOVJ C00198 BC00198 VJ=30.00
MOVJ C00199 BC00199 VJ=30.00
MOVL C00200 BC00200 V=500.0
'------------------------
'W63.20
'------------------------
SFTON P0308
MOVL C00201 BC00201 V=166.7 PL=0
ARCON
MOVL C00202 BC00202 V=10.0
ARCOF
MOVL C00203 BC00203 V=166.7 PL=0
SFTOF
COMM 'PRZEJAZD
COMM MOVL C00204 BC00204 V=500.0
COMM '------------------------
COMM 'W63.23
COMM '------------------------
COMM SFTON P0309
COMM MOVL C00205 BC00205 V=166.7 PL=0
COMM ARCON
COMM MOVL C00206 BC00206 V=10.0
COMM ARCOF
COMM MOVL C00207 BC00207 V=250.0 PL=0
COMM SFTOF
COMM MOVL C00208 BC00208 V=500.0
COMM SFTON P0310
COMM MOVL C00209 BC00209 V=166.7 PL=0
COMM ARCON
COMM MOVL C00210 BC00210 V=10.0
COMM ARCOF
COMM MOVL C00211 BC00211 V=250.0 PL=0
COMM SFTOF
MOVL C00212 BC00212 V=500.0
MOVL C00213 BC00213 V=500.0
MOVL C00214 BC00214 V=333.3
MOVL C00215 BC00215 V=250.0
'------------------------
'W29.29
'------------------------
SFTON P0312
MOVL C00216 BC00216 V=166.7 PL=0
ARCON
MOVL C00217 BC00217 V=9.2
ARCOF
MOVL C00218 BC00218 V=250.0 PL=0
MOVL C00219 BC00219 V=333.3
ARCON
MOVL C00220 BC00220 V=9.2
ARCOF
SFTOF
'PRZEJAZD
MOVL C00221 BC00221 V=333.3
MOVJ C00222 BC00222 VJ=30.00
MOVJ C00223 BC00223 VJ=20.00
MOVJ C00224 BC00224 VJ=50.00
MOVJ C00225 BC00225 VJ=20.00
MOVJ C00226 BC00226 VJ=10.00
MOVJ C00227 BC00227 VJ=20.00
MOVJ C00228 BC00228 VJ=20.00
'------------------------
'W28.2
'------------------------
MOVJ C00229 BC00229 VJ=10.00
MOVJ C00230 BC00230 VJ=10.00
MOVL C00231 BC00231 V=500.0
MOVL C00232 BC00232 V=500.0
'------------------------
'W62.5
'------------------------
SFTON P0351
MOVL C00233 BC00233 V=166.7 PL=0
ARCON
MOVL C00234 BC00234 V=10.0
ARCOF
MOVL C00235 BC00235 V=250.0 PL=0
SFTOF
'PRZEJAZD
MOVL C00236 BC00236 V=500.0
MOVL C00237 BC00237 V=500.0
MOVL C00238 BC00238 V=500.0
SFTON P0352
MOVL C00239 BC00239 V=166.7 PL=0
ARCON
MOVL C00240 BC00240 V=10.0
ARCOF
MOVL C00241 BC00241 V=250.0 PL=0
SFTOF
MOVL C00242 BC00242 V=500.0
'------------------------
'W29.8
'------------------------
SFTON P0353
MOVL C00243 BC00243 V=166.7 PL=0
ARCON
MOVL C00244 BC00244 V=10.0
ARCOF
MOVL C00245 BC00245 V=250.0 PL=0
SFTOF
MOVL C00246 BC00246 V=500.0
'PRZEJAZD
MOVL C00247 BC00247 V=500.0
MOVJ C00248 BC00248 VJ=20.00
MOVL C00249 BC00249 V=500.0
MOVL C00250 BC00250 V=500.0
MOVL C00251 BC00251 V=500.0
'------------------------
'W29.11
'------------------------
SFTON P0354
MOVL C00252 BC00252 V=166.7 PL=0
ARCON
MOVL C00253 BC00253 V=10.0
ARCOF
MOVL C00254 BC00254 V=250.0 PL=0
SFTOF
'PRZEJAZD
MOVL C00255 BC00255 V=500.0
'------------------------
'W29.14
'------------------------
SFTON P0355
MOVL C00256 BC00256 V=166.7 PL=0
ARCON
MOVL C00257 BC00257 V=10.0
ARCOF
MOVL C00258 BC00258 V=250.0 PL=0
SFTOF
'PRZEJAZD
MOVL C00259 BC00259 V=500.0
'------------------------
'W63.17
'------------------------
SFTON P0356
MOVL C00260 BC00260 V=166.7 PL=0
ARCON
MOVL C00261 BC00261 V=10.0
ARCOF
MOVL C00262 BC00262 V=250.0 PL=0
SFTOF
MOVL C00263 BC00263 V=500.0
SFTON P0357
MOVL C00264 BC00264 V=166.7 PL=0
ARCON
MOVL C00265 BC00265 V=10.0
ARCOF
MOVL C00266 BC00266 V=250.0 PL=0
SFTOF
'PRZEJAZD
MOVL C00267 BC00267 V=500.0
MOVJ C00268 BC00268 VJ=30.00
MOVJ C00269 BC00269 VJ=30.00
MOVJ C00270 BC00270 VJ=30.00
MOVL C00271 BC00271 V=500.0
MOVL C00272 BC00272 V=500.0
'------------------------
'W62.20
'------------------------
SFTON P0358
MOVL C00273 BC00273 V=166.7 PL=0
ARCON
MOVL C00274 BC00274 V=10.0
ARCOF
MOVL C00275 BC00275 V=250.0 PL=0
SFTOF
COMM 'PRZEJAZD
COMM MOVL C00276 BC00276 V=500.0
COMM '------------------------
COMM 'W63.23
COMM '------------------------
COMM SFTON P0359
COMM MOVL C00277 BC00277 V=166.7 PL=0
COMM ARCON
COMM MOVL C00278 BC00278 V=10.0
COMM ARCOF
COMM MOVL C00279 BC00279 V=250.0 PL=0
COMM MOVL C00280 BC00280 V=500.0
COMM '------------------------
COMM 'W29.29
COMM '------------------------
COMM SFTON P0360
COMM MOVL C00281 BC00281 V=166.7 PL=0
COMM ARCON
COMM MOVL C00282 BC00282 V=10.0
COMM ARCOF
COMM MOVL C00283 BC00283 V=250.0 PL=0
COMM SFTOF
COMM '------------------------
COMM 'W29.32
COMM '------------------------
COMM 'PRZEJAZD
MOVL C00284 BC00284 V=500.0
MOVJ C00285 BC00285 VJ=10.00
MOVL C00286 BC00286 V=416.7
SFTON P0362
MOVL C00287 BC00287 V=166.7 PL=0
ARCON
MOVL C00288 BC00288 V=9.2
ARCOF
MOVL C00289 BC00289 V=250.0 PL=0
MOVL C00290 BC00290 V=250.0
MOVL C00291 BC00291 V=166.7
ARCON
MOVL C00292 BC00292 V=9.2
ARCOF
SFTOF
MOVL C00293 BC00293 V=166.7
MOVJ C00294 BC00294 VJ=20.00
MOVJ C00295 BC00295 VJ=30.00
MOVJ C00296 BC00296 VJ=30.00
PAUSE
CALL JOB:MOVE_OUT_OF_TUNNEL
CALL JOB:CLEAN-R1
CALL JOB:MOVE_INTO_TUNNEL
'KONIEC SPAWANIA WEW STRONA
MOVJ C00297 BC00297 VJ=10.00
MOVJ C00298 BC00298 VJ=10.00
MOVJ C00299 BC00299 VJ=20.00
MOVJ C00300 BC00300 VJ=20.00
MOVJ C00301 BC00301 VJ=10.00
MOVJ C00302 BC00302 VJ=10.00
'------------------------
'W29.2
'------------------------
MOVL C00303 BC00303 V=500.0
'------------------------
'W63.5
'------------------------
SFTOF
MOVL C00304 BC00304 V=166.7 PL=0
REFP 3 C00305 BC00305
CALL JOB:SEARCH-R1
IMOV P0056 V=50.0 PL=0
SET P0301 P0006
SFTON P0301
REFP 3 C00306 BC00306
CALL JOB:SEARCH-R1
SET P0301 P0006
SFTON P0301
MOVL C00307 BC00307 V=166.7 PL=0
SFTOF
MOVL C00308 BC00308 V=500.0
MOVL C00309 BC00309 V=166.7 PL=0
REFP 3 C00310 BC00310
CALL JOB:SEARCH-R1
IMOV P0056 V=50.0 PL=0
SET P0302 P0006
SFTON P0302
REFP 3 C00311 BC00311
CALL JOB:SEARCH-R1
SET P0302 P0006
SFTON P0302
MOVL C00312 BC00312 V=166.7 PL=0
SFTOF
MOVL C00313 BC00313 V=500.0
MOVL C00314 BC00314 V=166.7 PL=0
REFP 3 C00315 BC00315
CALL JOB:SEARCH-R1
IMOV P0056 V=50.0 PL=0
SET P0303 P0006
SFTON P0303
REFP 3 C00316 BC00316
CALL JOB:SEARCH-R1
SET P0303 P0006
SFTON P0303
SFTOF
MOVL C00317 BC00317 V=166.7 PL=0
MOVL C00318 BC00318 V=500.0
MOVJ C00319 BC00319 VJ=30.00
MOVJ C00320 BC00320 VJ=30.00
MOVJ C00321 BC00321 VJ=20.00
MOVJ C00322 BC00322 VJ=30.00
MOVL C00323 BC00323 V=500.0
'------------------------
'W29.14
'------------------------
MOVL C00324 BC00324 V=166.7 PL=0
REFP 3 C00325 BC00325
CALL JOB:SEARCH-R1
IMOV P0056 V=23.0 PL=0
SET P0304 P0006
SFTON P0304
REFP 3 C00326 BC00326
CALL JOB:SEARCH-R1
SET P0304 P0006
SFTON P0304
MOVL C00327 BC00327 V=66.7 PL=0
SFTOF
'PRZEJAZD
MOVL C00328 BC00328 V=500.0
MOVL C00329 BC00329 V=500.0
'------------------------
'W63.17
'------------------------
MOVL C00330 BC00330 V=166.7 PL=0
REFP 3 C00331 BC00331
CALL JOB:SEARCH-R1
IMOV P0056 V=23.0 PL=0
SET P0305 P0006
SFTON P0305
REFP 3 C00332 BC00332
CALL JOB:SEARCH-R1
SET P0305 P0006
SFTON P0305
MOVL C00333 BC00333 V=166.7 PL=0
SFTOF
MOVL C00334 BC00334 V=500.0
MOVL C00335 BC00335 V=166.7
REFP 3 C00336 BC00336
CALL JOB:SEARCH-R1
IMOV P0056 V=23.0 PL=0
SET P0306 P0006
SFTON P0306
REFP 3 C00337 BC00337
CALL JOB:SEARCH-R1
SET P0306 P0006
SFTON P0306
MOVL C00338 BC00338 V=166.7 PL=0
'PRZEJAZD
MOVL C00339 BC00339 V=500.0
MOVL C00340 BC00340 V=166.7
REFP 3 C00341 BC00341
CALL JOB:SEARCH-R1
IMOV P0056 V=23.0 PL=0
SET P0307 P0006
SFTON P0307
REFP 3 C00342 BC00342
CALL JOB:SEARCH-R1
SET P0307 P0006
SFTON P0307
MOVL C00343 BC00343 V=166.7 PL=0
SFTOF
MOVJ C00344 BC00344 VJ=20.00
MOVJ C00345 BC00345 VJ=20.00
MOVJ C00346 BC00346 VJ=30.00
MOVJ C00347 BC00347 VJ=30.00
MOVL C00348 BC00348 V=500.0
'------------------------
'W63.20
'------------------------
MOVL C00349 BC00349 V=166.7 PL=0
REFP 3 C00350 BC00350
CALL JOB:SEARCH-R1
IMOV P0056 V=23.0 PL=0
SET P0308 P0006
SFTON P0308
REFP 3 C00351 BC00351
CALL JOB:SEARCH-R1
SET P0308 P0006
SFTON P0308
MOVL C00352 BC00352 V=166.7 PL=0
SFTOF
COMM 'PRZEJAZD
COMM MOVL C00353 BC00353 V=500.0
COMM '------------------------
COMM 'W63.23
COMM '------------------------
COMM MOVL C00354 BC00354 V=166.7 PL=0
COMM REFP 3 C00355 BC00355
COMM CALL JOB:SEARCH-R1
COMM IMOV P0056 V=23.0 PL=0
COMM SET P0309 P0006
COMM SFTON P0309
COMM REFP 3 C00356 BC00356
COMM CALL JOB:SEARCH-R1
COMM SET P0309 P0006
COMM SFTON P0309
COMM MOVL C00357 BC00357 V=250.0 PL=0
COMM SFTOF
COMM MOVL C00358 BC00358 V=500.0
COMM MOVL C00359 BC00359 V=166.7 PL=0
COMM REFP 3 C00360 BC00360
COMM CALL JOB:SEARCH-R1
COMM IMOV P0056 V=23.0 PL=0
COMM SET P0310 P0006
COMM SFTON P0310
COMM REFP 3 C00361 BC00361
COMM CALL JOB:SEARCH-R1
COMM SET P0310 P0006
COMM SFTON P0310
COMM MOVL C00362 BC00362 V=250.0 PL=0
COMM SFTOF
MOVL C00363 BC00363 V=500.0
MOVL C00364 BC00364 V=500.0
MOVL C00365 BC00365 V=500.0
MOVL C00366 BC00366 V=333.3
'------------------------
'W29.29
'------------------------
MOVL C00367 BC00367 V=250.0
MOVL C00368 BC00368 V=166.7 PL=0
REFP 3 C00369 BC00369
CALL JOB:SEARCH-R1
IMOV P0056 V=23.0 PL=0
SET P0312 P0006
SFTON P0312
REFP 3 C00370 BC00370
CALL JOB:SEARCH-R1
SET P0312 P0006
SFTON P0312
MOVL C00371 BC00371 V=250.0 PL=0
SFTOF
'PRZEJAZD
MOVL C00372 BC00372 V=333.3
'PRZEJAZD
MOVJ C00373 BC00373 VJ=20.00
MOVJ C00374 BC00374 VJ=50.00
MOVJ C00375 BC00375 VJ=20.00
MOVJ C00376 BC00376 VJ=10.00
'------------------------
'W28.2
'------------------------
MOVJ C00377 BC00377 VJ=10.00
MOVJ C00378 BC00378 VJ=10.00
MOVL C00379 BC00379 V=500.0
MOVL C00380 BC00380 V=500.0
'------------------------
'W62.5
'------------------------
MOVL C00381 BC00381 V=166.7 PL=0
REFP 3 C00382 BC00382
CALL JOB:SEARCH-R1
IMOV P0056 V=23.0 PL=0
SET P0351 P0006
SFTON P0351
REFP 3 C00383 BC00383
CALL JOB:SEARCH-R1
SET P0351 P0006
SFTON P0351
MOVL C00384 BC00384 V=250.0 PL=0
SFTOF
'PRZEJAZD
MOVL C00385 BC00385 V=500.0
MOVL C00386 BC00386 V=500.0
MOVL C00387 BC00387 V=500.0
MOVL C00388 BC00388 V=166.7 PL=0
REFP 3 C00389 BC00389
CALL JOB:SEARCH-R1
IMOV P0056 V=23.0 PL=0
SET P0352 P0006
SFTON P0352
REFP 3 C00390 BC00390
CALL JOB:SEARCH-R1
SET P0352 P0006
SFTON P0352
MOVL C00391 BC00391 V=250.0 PL=0
SFTOF
MOVL C00392 BC00392 V=500.0
'------------------------
'W29.8
'------------------------
MOVL C00393 BC00393 V=166.7 PL=0
REFP 3 C00394 BC00394
CALL JOB:SEARCH-R1
IMOV P0056 V=23.0 PL=0
SET P0353 P0006
SFTON P0353
REFP 3 C00395 BC00395
CALL JOB:SEARCH-R1
SET P0353 P0006
SFTON P0353
MOVL C00396 BC00396 V=250.0 PL=0
SFTOF
MOVL C00397 BC00397 V=500.0
'PRZEJAZD
MOVL C00398 BC00398 V=500.0
MOVJ C00399 BC00399 VJ=20.00
MOVJ C00400 BC00400 VJ=20.00
MOVL C00401 BC00401 V=500.0
MOVL C00402 BC00402 V=500.0
MOVL C00403 BC00403 V=500.0
'------------------------
'W29.11
'------------------------
MOVL C00404 BC00404 V=166.7 PL=0
REFP 3 C00405 BC00405
CALL JOB:SEARCH-R1
IMOV P0056 V=23.0 PL=0
SET P0354 P0006
SFTON P0354
REFP 3 C00406 BC00406
CALL JOB:SEARCH-R1
SET P0354 P0006
SFTON P0354
MOVL C00407 BC00407 V=250.0 PL=0
SFTOF
'PRZEJAZD
MOVL C00408 BC00408 V=500.0
'------------------------
'W29.14
'------------------------
MOVL C00409 BC00409 V=166.7 PL=0
REFP 3 C00410 BC00410
CALL JOB:SEARCH-R1
IMOV P0056 V=23.0 PL=0
SET P0355 P0006
SFTON P0355
REFP 3 C00411 BC00411
CALL JOB:SEARCH-R1
SET P0355 P0006
SFTON P0355
MOVL C00412 BC00412 V=250.0 PL=0
SFTOF
'PRZEJAZD
MOVL C00413 BC00413 V=500.0
'------------------------
'W63.17
'------------------------
MOVL C00414 BC00414 V=166.7 PL=0
REFP 3 C00415 BC00415
CALL JOB:SEARCH-R1
IMOV P0056 V=23.0 PL=0
SET P0356 P0006
SFTON P0356
REFP 3 C00416 BC00416
CALL JOB:SEARCH-R1
SET P0356 P0006
SFTON P0356
MOVL C00417 BC00417 V=250.0 PL=0
SFTOF
MOVL C00418 BC00418 V=500.0
MOVL C00419 BC00419 V=166.7 PL=0
REFP 3 C00420 BC00420
CALL JOB:SEARCH-R1
IMOV P0056 V=23.0 PL=0
SET P0357 P0006
SFTON P0357
REFP 3 C00421 BC00421
CALL JOB:SEARCH-R1
SET P0357 P0006
SFTON P0357
MOVL C00422 BC00422 V=250.0 PL=0
SFTOF
'PRZEJAZD
MOVL C00423 BC00423 V=500.0
MOVJ C00424 BC00424 VJ=30.00
MOVJ C00425 BC00425 VJ=30.00
MOVL C00426 BC00426 V=500.0
MOVL C00427 BC00427 V=500.0
'------------------------
'W62.20
'------------------------
MOVL C00428 BC00428 V=166.7 PL=0
REFP 3 C00429 BC00429
CALL JOB:SEARCH-R1
IMOV P0056 V=23.0 PL=0
SET P0358 P0006
SFTON P0358
REFP 3 C00430 BC00430
CALL JOB:SEARCH-R1
SET P0358 P0006
SFTON P0358
MOVL C00431 BC00431 V=250.0 PL=0
SFTOF
COMM 'PRZEJAZD
COMM MOVL C00432 BC00432 V=500.0
COMM '------------------------
COMM 'W63.23
COMM '------------------------
COMM MOVL C00433 BC00433 V=166.7 PL=0
COMM REFP 3 C00434 BC00434
COMM CALL JOB:SEARCH-R1
COMM IMOV P0056 V=23.0 PL=0
COMM SET P0359 P0006
COMM SFTON P0359
COMM REFP 3 C00435 BC00435
COMM CALL JOB:SEARCH-R1
COMM SET P0359 P0006
COMM SFTON P0359
COMM MOVL C00436 BC00436 V=250.0 PL=0
COMM MOVL C00437 BC00437 V=500.0
COMM '------------------------
COMM 'W29.29
COMM '------------------------
COMM MOVL C00438 BC00438 V=166.7 PL=0
COMM REFP 3 C00439 BC00439
COMM CALL JOB:SEARCH-R1
COMM IMOV P0056 V=23.0 PL=0
COMM SET P0360 P0006
COMM SFTON P0360
COMM REFP 3 C00440 BC00440
COMM CALL JOB:SEARCH-R1
COMM SET P0360 P0006
COMM SFTON P0360
COMM MOVL C00441 BC00441 V=250.0 PL=0
COMM SFTOF
COMM 'PRZEJAZD
COMM SFTOF
COMM '------------------------
COMM 'W29.32
COMM '------------------------
COMM 'PRZEJAZD
MOVL C00442 BC00442 V=500.0
MOVL C00443 BC00443 V=500.0
MOVL C00444 BC00444 V=416.7
MOVL C00445 BC00445 V=166.7 PL=0
REFP 3 C00446 BC00446
CALL JOB:SEARCH-R1
IMOV P0056 V=23.0 PL=0
SET P0362 P0006
SFTON P0362
REFP 3 C00447 BC00447
CALL JOB:SEARCH-R1
SET P0362 P0006
SFTON P0362
MOVL C00448 BC00448 V=250.0 PL=0
SFTOF
MOVJ C00449 BC00449 VJ=20.00
MOVJ C00450 BC00450 VJ=30.00
MOVJ C00451 BC00451 VJ=30.00
'KONIEC SEARCH WEW STRONA
MOVJ C00452 BC00452 VJ=30.00
MOVJ C00453 BC00453 VJ=20.00
MOVJ C00454 BC00454 VJ=10.00
MOVJ C00455 BC00455 VJ=20.00
MOVJ C00456 BC00456 VJ=20.00
'------------------------
'W29.2
'------------------------
MOVL C00457 BC00457 V=500.0
'------------------------
'W63.5
MACRO1 MJ#(0) ARGF9
'------------------------
SFTOF
SFTON P0301
MOVL C00458 BC00458 V=166.7 PL=0
ARCON
MOVL C00459 BC00459 V=8.3
ARCOF
SFTOF
MOVL C00460 BC00460 V=500.0
MACRO1 MJ#(0) ARGF24
SFTON P0302
MOVL C00461 BC00461 V=166.7 PL=0
ARCON
MOVL C00462 BC00462 V=8.3
ARCOF
MOVL C00463 BC00463 V=166.7 PL=0
SFTOF
MOVL C00464 BC00464 V=500.0
SFTON P0303
MOVL C00465 BC00465 V=166.7 PL=0
ARCON
MOVL C00466 BC00466 V=8.3
ARCOF
SFTOF
MOVL C00467 BC00467 V=166.7 PL=0
MOVL C00468 BC00468 V=500.0
MOVJ C00469 BC00469 VJ=30.00
MOVJ C00470 BC00470 VJ=20.00
MOVJ C00471 BC00471 VJ=30.00
MOVJ C00472 BC00472 VJ=30.00
MOVL C00473 BC00473 V=500.0
'------------------------
'W29.14
'------------------------
SFTON P0304
MOVL C00474 BC00474 V=166.7 PL=0
ARCON
MOVL C00475 BC00475 V=8.3
ARCOF
MOVL C00476 BC00476 V=166.7 PL=0
SFTOF
'PRZEJAZD
MOVL C00477 BC00477 V=500.0
MOVL C00478 BC00478 V=500.0
'------------------------
'W63.17
'------------------------
SFTON P0305
MOVL C00479 BC00479 V=166.7 PL=0
ARCON
MOVL C00480 BC00480 V=8.3
ARCOF
MOVL C00481 BC00481 V=166.7 PL=0
SFTOF
MOVL C00482 BC00482 V=500.0
SFTON P0306
MOVL C00483 BC00483 V=166.7
ARCON
MOVL C00484 BC00484 V=8.3
ARCOF
MOVL C00485 BC00485 V=166.7 PL=0
SFTOF
'PRZEJAZD
MOVL C00486 BC00486 V=500.0
SFTON P0307
MOVL C00487 BC00487 V=166.7
ARCON
MOVL C00488 BC00488 V=8.3
ARCOF
MOVL C00489 BC00489 V=166.7 PL=0
SFTOF
MOVJ C00490 BC00490 VJ=20.00
MOVJ C00491 BC00491 VJ=20.00
MOVJ C00492 BC00492 VJ=30.00
MOVJ C00493 BC00493 VJ=30.00
MOVL C00494 BC00494 V=500.0
'------------------------
'W63.20
'------------------------
SFTON P0308
MOVL C00495 BC00495 V=166.7 PL=0
ARCON
MOVL C00496 BC00496 V=8.3
ARCOF
MOVL C00497 BC00497 V=166.7 PL=0
SFTOF
COMM 'PRZEJAZD
COMM MOVL C00498 BC00498 V=500.0
COMM '------------------------
COMM 'W63.23
COMM '------------------------
COMM SFTON P0309
COMM MOVL C00499 BC00499 V=166.7 PL=0
COMM ARCON
COMM MOVL C00500 BC00500 V=8.3
COMM ARCOF
COMM MOVL C00501 BC00501 V=250.0 PL=0
COMM SFTOF
COMM MOVL C00502 BC00502 V=500.0
COMM SFTON P0310
COMM MOVL C00503 BC00503 V=166.7 PL=0
COMM ARCON
COMM MOVL C00504 BC00504 V=8.3
COMM ARCOF
COMM MOVL C00505 BC00505 V=250.0 PL=0
COMM SFTOF
MOVL C00506 BC00506 V=500.0
MOVL C00507 BC00507 V=500.0
MOVL C00508 BC00508 V=333.3
'------------------------
'W29.29
'------------------------
MOVL C00509 BC00509 V=500.0
SFTON P0312
MOVL C00510 BC00510 V=166.7 PL=0
ARCON
MOVL C00511 BC00511 V=8.3
ARCOF
MOVL C00512 BC00512 V=250.0 PL=0
MOVL C00513 BC00513 V=500.0
MOVL C00514 BC00514 V=166.7
ARCON
MOVL C00515 BC00515 V=8.3
ARCOF
SFTOF
'PRZEJAZD
MOVL C00516 BC00516 V=333.3
'PRZEJAZD
'KONIEC SPAWANIA CZESCI WSPOLNEJ
MOVJ C00517 BC00517 VJ=20.00
MOVJ C00518 BC00518 VJ=50.00
MOVJ C00519 BC00519 VJ=20.00
MOVJ C00520 BC00520 VJ=10.00
MOVJ C00521 BC00521 VJ=20.00
MOVJ C00522 BC00522 VJ=20.00
'------------------------
'W28.2
'------------------------
MOVJ C00523 BC00523 VJ=10.00
MOVJ C00524 BC00524 VJ=10.00
MOVL C00525 BC00525 V=500.0
MOVL C00526 BC00526 V=500.0
'------------------------
'W62.5
'------------------------
SFTON P0351
MOVL C00527 BC00527 V=166.7 PL=0
ARCON
MOVL C00528 BC00528 V=8.3
ARCOF
MOVL C00529 BC00529 V=250.0 PL=0
SFTOF
'PRZEJAZD
MOVL C00530 BC00530 V=500.0
MOVL C00531 BC00531 V=500.0
MOVL C00532 BC00532 V=500.0
SFTON P0352
MOVL C00533 BC00533 V=166.7 PL=0
ARCON
MOVL C00534 BC00534 V=8.3
ARCOF
MOVL C00535 BC00535 V=250.0 PL=0
SFTOF
MOVL C00536 BC00536 V=500.0
'------------------------
'W29.8
'------------------------
SFTON P0353
MOVL C00537 BC00537 V=166.7 PL=0
ARCON
MOVL C00538 BC00538 V=8.3
ARCOF
MOVL C00539 BC00539 V=250.0 PL=0
SFTOF
MOVL C00540 BC00540 V=500.0
'PRZEJAZD
MOVL C00541 BC00541 V=500.0
MOVJ C00542 BC00542 VJ=20.00
MOVL C00543 BC00543 V=500.0
MOVL C00544 BC00544 V=500.0
MOVL C00545 BC00545 V=500.0
'------------------------
'W29.11
'------------------------
SFTON P0354
MOVL C00546 BC00546 V=166.7 PL=0
ARCON
MOVL C00547 BC00547 V=8.3
ARCOF
MOVL C00548 BC00548 V=250.0 PL=0
SFTOF
'PRZEJAZD
MOVL C00549 BC00549 V=500.0
'------------------------
'W29.14
'------------------------
SFTON P0355
MOVL C00550 BC00550 V=166.7 PL=0
ARCON
MOVL C00551 BC00551 V=8.3
ARCOF
MOVL C00552 BC00552 V=250.0 PL=0
SFTOF
'PRZEJAZD
MOVL C00553 BC00553 V=500.0
'------------------------
'W63.17
'------------------------
SFTON P0356
MOVL C00554 BC00554 V=166.7 PL=0
ARCON
MOVL C00555 BC00555 V=8.3
ARCOF
MOVL C00556 BC00556 V=250.0 PL=0
SFTOF
MOVL C00557 BC00557 V=500.0
SFTON P0357
MOVL C00558 BC00558 V=166.7 PL=0
ARCON
MOVL C00559 BC00559 V=8.3
ARCOF
MOVL C00560 BC00560 V=250.0 PL=0
SFTOF
'PRZEJAZD
MOVL C00561 BC00561 V=500.0
MOVJ C00562 BC00562 VJ=30.00
MOVJ C00563 BC00563 VJ=30.00
MOVJ C00564 BC00564 VJ=30.00
MOVL C00565 BC00565 V=500.0
MOVL C00566 BC00566 V=500.0
'------------------------
'W62.20
'------------------------
SFTON P0358
MOVL C00567 BC00567 V=166.7 PL=0
ARCON
MOVL C00568 BC00568 V=8.3
ARCOF
MOVL C00569 BC00569 V=250.0 PL=0
SFTOF
COMM 'PRZEJAZD
COMM MOVL C00570 BC00570 V=500.0
COMM '------------------------
COMM 'W63.23
COMM '------------------------
COMM SFTON P0359
COMM MOVL C00571 BC00571 V=166.7 PL=0
COMM ARCON
COMM MOVL C00572 BC00572 V=8.3
COMM ARCOF
COMM MOVL C00573 BC00573 V=250.0 PL=0
COMM MOVL C00574 BC00574 V=500.0
COMM '------------------------
COMM 'W29.29
COMM '------------------------
COMM SFTON P0360
COMM MOVL C00575 BC00575 V=166.7 PL=0
COMM ARCON
COMM MOVL C00576 BC00576 V=8.3
COMM ARCOF
COMM MOVL C00577 BC00577 V=250.0 PL=0
COMM SFTOF
COMM '------------------------
COMM 'W29.32
COMM '------------------------
COMM 'PRZEJAZD
MOVL C00578 BC00578 V=500.0
MOVL C00579 BC00579 V=500.0
MOVL C00580 BC00580 V=416.7
MOVL C00581 BC00581 V=500.0
SFTON P0362
MOVL C00582 BC00582 V=166.7 PL=0
ARCON
MOVL C00583 BC00583 V=8.3
ARCOF
MOVL C00584 BC00584 V=250.0 PL=0
MOVL C00585 BC00585 V=500.0
MOVL C00586 BC00586 V=166.7
ARCON
MOVL C00587 BC00587 V=8.3
ARCOF
MOVL C00588 BC00588 V=250.0
SFTOF
MOVJ C00589 BC00589 VJ=20.00
MOVJ C00590 BC00590 VJ=30.00
MOVJ C00591 BC00591 VJ=30.00
MOVJ C00592 BC00592 VJ=30.00
CALL JOB:MOVE_OUT_OF_TUNNEL
END
